Universal Robots PolyScope program: tt.urp

Program tt (installation=default directory=/programs/usbdisk createdIn=5.18.0 lastSavedIn=5.18.0 robotSerialNumber=20245388888)
Calibrated DH parameters: a=[0, -0.24355, -0.2132, 0, 0, 0]; d=[0.15185, 0, 0, 0.13105, 0.08535, 0.0921]; alpha=[1.570796, 0, 0, 1.570796, -1.570796, 0]; deltaTheta=[0, 0, 0, 0, 0, 0]
InitVariablesNode
Robot Program (runOnlyOnce=false)
  MoveL speed 250 mm/s, acceleration 1200 mm/s^2 (useActiveTCP=true optimoveEnabled=true optiMovePercentage=30) feature=Base
    Waypoint base: TCP in base x=-339.797 y=122.56 z=472.551 mm, rx=-1.0316 ry=-1.2454 rz=1.141 rad; joints [181.364, -176.166, 84.116, 275.907, 90.27, -9.076] deg
  MoveL speed 250 mm/s, acceleration 1200 mm/s^2 (useActiveTCP=true optimoveEnabled=true optiMovePercentage=30) feature=Joint_6_name
    Waypoint tool: TCP in base x=-339.797 y=122.56 z=472.551 mm, rx=-1.0316 ry=-1.2454 rz=1.141 rad; joints [181.364, -176.166, 84.116, 275.907, 90.27, -9.076] deg; feature pose in base x=-339.821 y=122.543 z=472.539 mm, rx=-1.0316 ry=-1.2455 rz=1.141 rad
  Wait Sleep waitTime=1
  MoveL speed 250 mm/s, acceleration 1200 mm/s^2 (useActiveTCP=true optimoveEnabled=false optiMovePercentage=30) feature=Base
    Waypoint Waypoint_4: TCP in base x=-339.796 y=122.576 z=472.553 mm, rx=-1.0316 ry=-1.2453 rz=1.141 rad; joints [181.362, -176.165, 84.114, 275.907, 90.268, -9.075] deg; TCP offset x=0 y=0 z=0 mm, rx=0 ry=0 rz=0 rad
    Waypoint Waypoint_3: TCP in base x=-339.797 y=122.56 z=472.551 mm, rx=-1.0316 ry=-1.2454 rz=1.141 rad; joints [181.364, -176.166, 84.116, 275.907, 90.27, -9.076] deg
